(* PLC project 01_Pulsador_Lampara.project, CODESYS CODESYS V3.5 SP22 Patch 3 *)
(* stored: creationDateTime 2026-08-12T12:51:23.0960455, modificationDateTime 2026-08-11T17:53:31.5723282 *)

PROGRAM PLC_PRG
  VAR
    xPulsador : BOOL;
    xLampara : BOOL;
  END_VAR

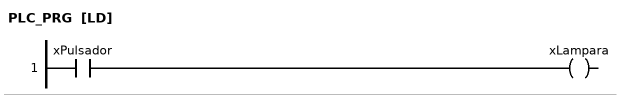
(* LD diagram, written out as Structured Text *)

xLampara := xPulsador;
END_PROGRAM

CONFIGURATION Device
  RESOURCE Application ON PLC
    TASK MainTask(INTERVAL := T#20ms, PRIORITY := 1);
    PROGRAM PLC_PRG WITH MainTask : PLC_PRG;
  END_RESOURCE
END_CONFIGURATION
